{region '#Template'}
	{attribute 'Version' := '1.2.1.0'}
	{attribute 'Tags' := '"LCID": "1031", "Text": "Universal, Control, Trend"'}
	{attribute 'Tags' := '"LCID": "1033", "Text": "Universal, Control, Trend"'}
	{attribute 'Using' := '"Type": "Template", "URI": "EC_AMEV"'}
	{attribute 'Using' := '"Type": "Template", "URI": "BA2_Param"'}
	{attribute 'Description' := '"LCID": "1031", "Text": "Trend"'}
	{attribute 'Description' := '"LCID": "1033", "Text": "Trend"'}
{endregion}			 
FUNCTION_BLOCK FB_BA_TrendLogging EXTENDS FB_BA_View
VAR_INPUT
END_VAR
VAR_OUTPUT
END_VAR
VAR_INPUT CONSTANT
	Trends						: ARRAY[1..TREND_COUNT] OF FB_BA_Trend;								
END_VAR
VAR
	i							: UDINT;
END_VAR
VAR CONSTANT
	TREND_COUNT						: UDINT := 30;
END_VAR

SUPER^();

FOR i := 1 TO TREND_COUNT DO
	Trends[i]();
END_FOR

METHOD FB_init : BOOL
VAR_INPUT
	bInitRetains : BOOL; // if TRUE, the retain variables are initialized (warm start / cold start)
	bInCopyCode : BOOL;  // if TRUE, the instance afterwards gets moved into the copy code (online change)
END_VAR 
VAR
	sIdx	: STRING;
END_VAR
FOR i := 1 TO TREND_COUNT DO
	sIdx := CONCAT(TO_STRING(i),'}');;

	Trends[i].iParent					:= THIS^;
	Trends[i].iLabel					:= LblFunctions_ObjectTrendLog;
	Trends[i].sObjectName				:= CONCAT('{Idx=',sIdx);
	Trends[i].bEnable					:= BA2_Param.bTrend_DefLogEnable;
	Trends[i].stStartTime				:= BA2_Param.stTrend_DefStartTime;
	Trends[i].stStopTime				:= BA2_Param.stTrend_DefStopTime;	
	Trends[i].nLogInterval 				:= BA2_Param.nTrend_DefLogInterval;
	Trends[i].bStopOnFull				:= BA2_Param.bTrend_DefStopOnFull;
	Trends[i].nBufferSize 				:= BA2_Param.nTrend_BufferSize;
	Trends[i].eLoggingType				:= BA2_Param.eTrend_DefLoggingType;	
	Trends[i].nEventClassID				:= EC_ID.NC80;
	Trends[i].nNotificationThreshold	:= BA2_Param.nTrend_DefNotificationThreshold;
	Trends[i].aEventTransitionText[1]	:= txtEvent_Offnormal;
	Trends[i].aEventTransitionText[2]	:= txtEvent_None;
	Trends[i].aEventTransitionText[3]	:= txtEvent_Normal;
	Trends[i].bEventDetectionEnable		:= FALSE;
	Trends[i].aEventEnable[1]			:= TRUE;			//	to_offnormal
	Trends[i].aEventEnable[2]			:= TRUE;			//	to_fault
	Trends[i].aEventEnable[3]			:= TRUE;			//	to_normal	
	Trends[i].bAcknowledgeRm			:= FALSE;		
END_FOR
END_METHOD

END_FUNCTION_BLOCK

(* stored: Version 1.1.0.1, ProductVersion 3.1.4024.9
   POU FB_BA_TrendLogging: Id {c66a71d4-cea6-4416-8e55-61cc71db2e16}, SpecialFunc None
   Method FB_init: Id {0b7f1b57-d8a3-4221-aa2c-f2c7e43f1646} *)
